(* Logix 5000 project; controller R5_CSS vendor 1 type 14 code 74 rev 19.11; software revision 19.01; part 18 of 18 *)
(* tags used below, declared in another part *)
   AlarmMasterDisable : BOOL;
   AutoTune : PIDE_AUTOTUNE;
   CSS_Heartbeat : BOOL;
   CSS_HeartbeatOffONS : BOOL;
   CSS_HeartbeatOnONS : BOOL;
   CSS_OK_TO_RUN : BOOL;   // PRU_RUN_DISABLE 0 = Cannot Run 1 = OK to Run
   CSS_Status_To_UTL_Comms : DINT;
   Fault : BOOL;
   FC101 : FLOW_CONTROL;   // QUENCH BASIN FLOW TRANSMITTER CONTROL
   FC101_Initialize : BOOL;
   FC101_Initialize_TON : TIMER;
   FC140 : FLOW_CONTROL;
   FC140A : FLOW_CONTROL;   // QUENCH TOWER UPPER SPRAY FLOW CONTROL
   FC140B : FLOW_CONTROL;   // QUENCH TOWER LOWER SPRAY FLOW CONTROL
   FC365 : FLOW_CONTROL;   // COALESCER PROCESS IMPURITY FLOW CONTROL
   FT140_TOTAL_FLOW : REAL;
   InputMax_IF8 : REAL;
   InputMin_IF8 : REAL;
   LC101 : LEVEL_CONTROL;   // QUENCH TOWER BASIN LIT
   LC101_PIDE_AUTO : BOOL;
   LC101_PIDE_CV_Hold : REAL;
   LC303A : LEVEL_CONTROL;   // AQUEOUS PHASE OF PRIMARY SETTLER
   MSG_ConnectionRateSec : DINT;
   MSG_TimeoutMultiplier : DINT;
   MSG_UnconnectedTimeoutSec : DINT;
   MyTime : DINT[10];
   P303A : PUMP_CONTROL;
   P303B : PUMP_CONTROL;
   PC132 : PRESSURE_CONTROL;
   PC132_PID : PID;
   PID_FCV365 : PID;
   PID_TCV108_Flow : PID;
   PRU_BLOWER_SEQ : INT;   // PRU BLOWER SEQUENCE NUMBER
   PRU_Quantity : DINT;
   PRU_SEQ_TMR : TIMER;   // PRU_SEQUENCE TIMER
   PRUA_READ : INT[30];
   PRUB_READ : INT[30];
   PRUC_READ : INT[30];
   PRUD_READ : INT[30];   // PRU D READ
   PRUE_READ : INT[30];
   PRUF_READ : INT[30];
   PRUG_READ : INT[30];
   PRUH_READ : INT[30];
   RandomNumber : REAL;
   RandomNumberDint : DINT;
   TC108 : TEMP_CONTROL;   // QUENCH TOWER EXIT GAS TEMPERATURE CONTROL
   TestyBit : DINT;
   TIMER : TIMER[50];   // HX A TIMER FOR START
   UTIL_1 : INT;   // ONE SHOTS FOR UTILITIES
   UTL_AlarmMaster : DINT;
   UTL_Comms : DINT[3];
   UTL_CommsLossAlm : BOOL;
   UTL_HeartbeatTimer : TIMER;
   UTL_READ_MSG : MESSAGE;
   WRS_OK : BOOL;
(* MainProgram, continued *)

ROUTINE TEMPORARY   (* ladder *)
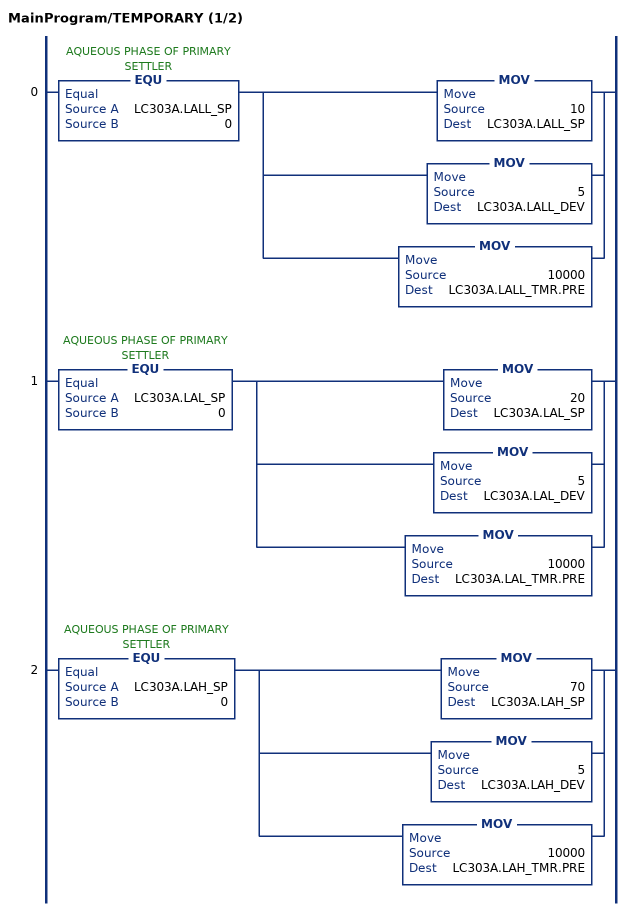
   0: EQU(LC303A.LALL_SP,0)[MOV(10,LC303A.LALL_SP) ,MOV(5,LC303A.LALL_DEV) ,MOV(10000,LC303A.LALL_TMR.PRE) ];
   1: EQU(LC303A.LAL_SP,0)[MOV(20,LC303A.LAL_SP) ,MOV(5,LC303A.LAL_DEV) ,MOV(10000,LC303A.LAL_TMR.PRE) ];
   2: EQU(LC303A.LAH_SP,0)[MOV(70,LC303A.LAH_SP) ,MOV(5,LC303A.LAH_DEV) ,MOV(10000,LC303A.LAH_TMR.PRE) ];
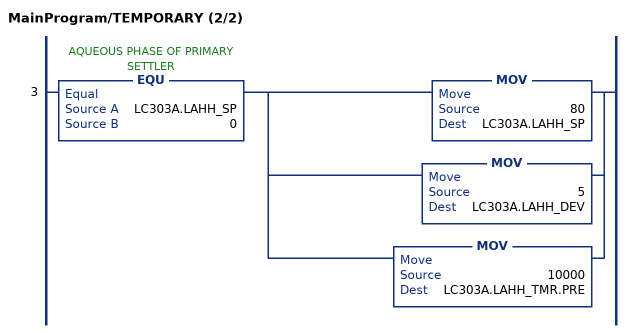
   3: EQU(LC303A.LAHH_SP,0)[MOV(80,LC303A.LAHH_SP) ,MOV(5,LC303A.LAHH_DEV) ,MOV(10000,LC303A.LAHH_TMR.PRE) ];
END_ROUTINE

ROUTINE UTIL   (* ladder *)
// UTILITIES LOGIC
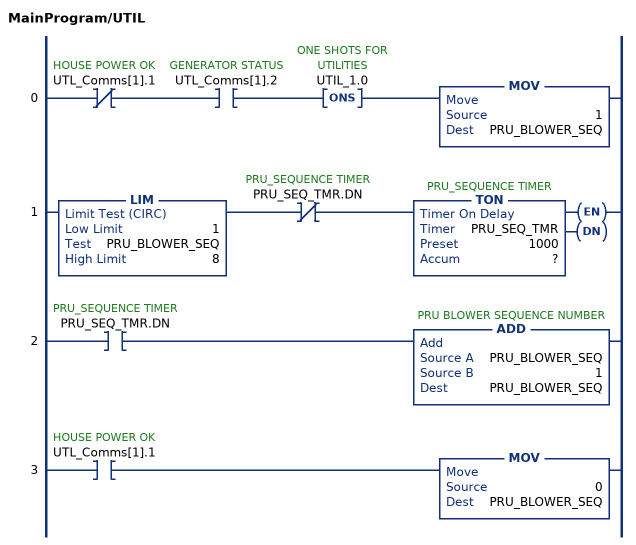
   0: XIO(UTL_Comms[1].1)XIC(UTL_Comms[1].2)ONS(UTIL_1.0)MOV(1,PRU_BLOWER_SEQ);
   1: LIM(1,PRU_BLOWER_SEQ,8)XIO(PRU_SEQ_TMR.DN)TON(PRU_SEQ_TMR,?,?);
   2: XIC(PRU_SEQ_TMR.DN)ADD(PRU_BLOWER_SEQ,1,PRU_BLOWER_SEQ);
   3: XIC(UTL_Comms[1].1)MOV(0,PRU_BLOWER_SEQ);
END_ROUTINE
END_PROGRAM

PROGRAM Never_Fault_Logic   (* main routine Main *)
VAR
   HMI_CONTROLLER_DISPLAY : MAJOR_FAULT := (TYPE := 3, CODE := 23);
   MAJORFAULT_RECORD : FAULTRECORD;
END_VAR

ROUTINE Main   (* ladder *)
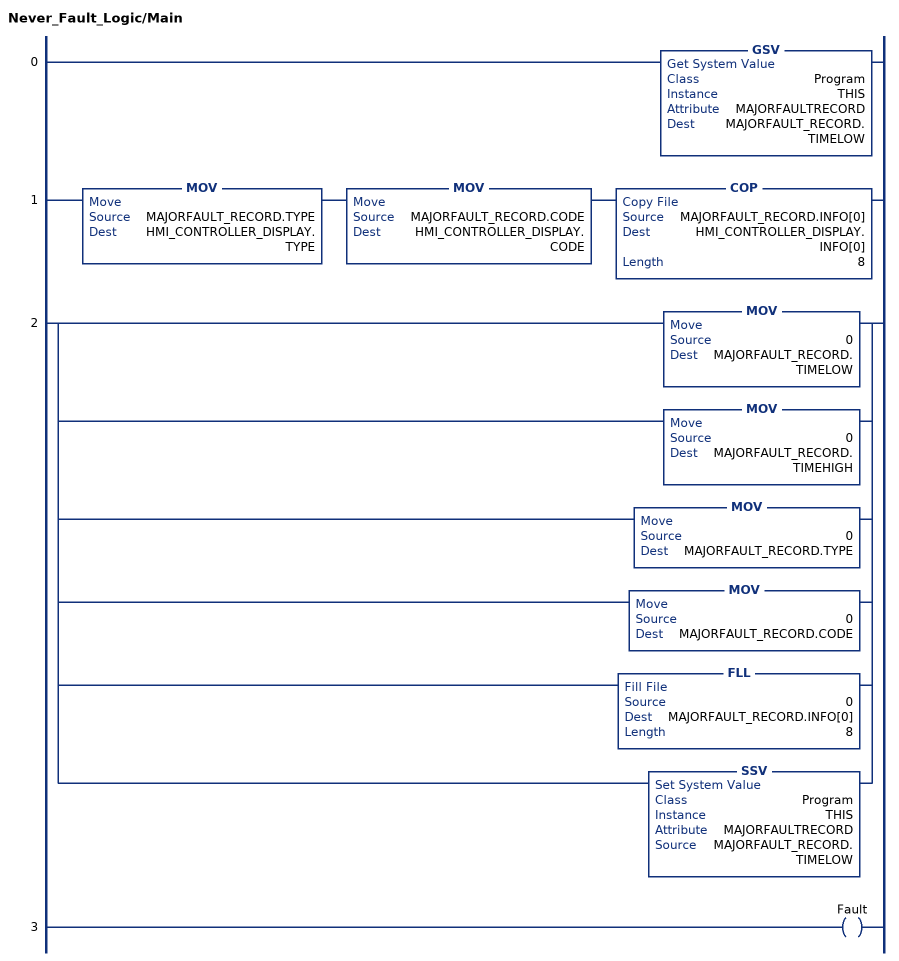
   0: GSV(Program,THIS,MAJORFAULTRECORD,MAJORFAULT_RECORD.TIMELOW);
   1: MOV(MAJORFAULT_RECORD.TYPE,HMI_CONTROLLER_DISPLAY.TYPE)MOV(MAJORFAULT_RECORD.CODE,HMI_CONTROLLER_DISPLAY.CODE)COP(MAJORFAULT_RECORD.INFO[0],HMI_CONTROLLER_DISPLAY.INFO[0],8);
   2: [MOV(0,MAJORFAULT_RECORD.TIMELOW) ,MOV(0,MAJORFAULT_RECORD.TIMEHIGH) ,MOV(0,MAJORFAULT_RECORD.TYPE) ,MOV(0,MAJORFAULT_RECORD.CODE) ,FLL(0,MAJORFAULT_RECORD.INFO[0],8) ,SSV(Program,THIS,MAJORFAULTRECORD,MAJORFAULT_RECORD.TIMELOW) ];
   3: OTE(Fault);
END_ROUTINE
END_PROGRAM

PROGRAM PIDE   (* main routine Main *)
VAR
   BNOT_01 : FBD_BOOLEAN_NOT := (Out := 1);
   BNOT_02 : FBD_BOOLEAN_NOT := (In := 1);
   SUB_01 : FBD_MATH := (SourceA := 0.049999237, SourceB := 29.966267, Dest := -29.916267);
END_VAR

ROUTINE LC101   (* function block diagram *)
   SHEET 1
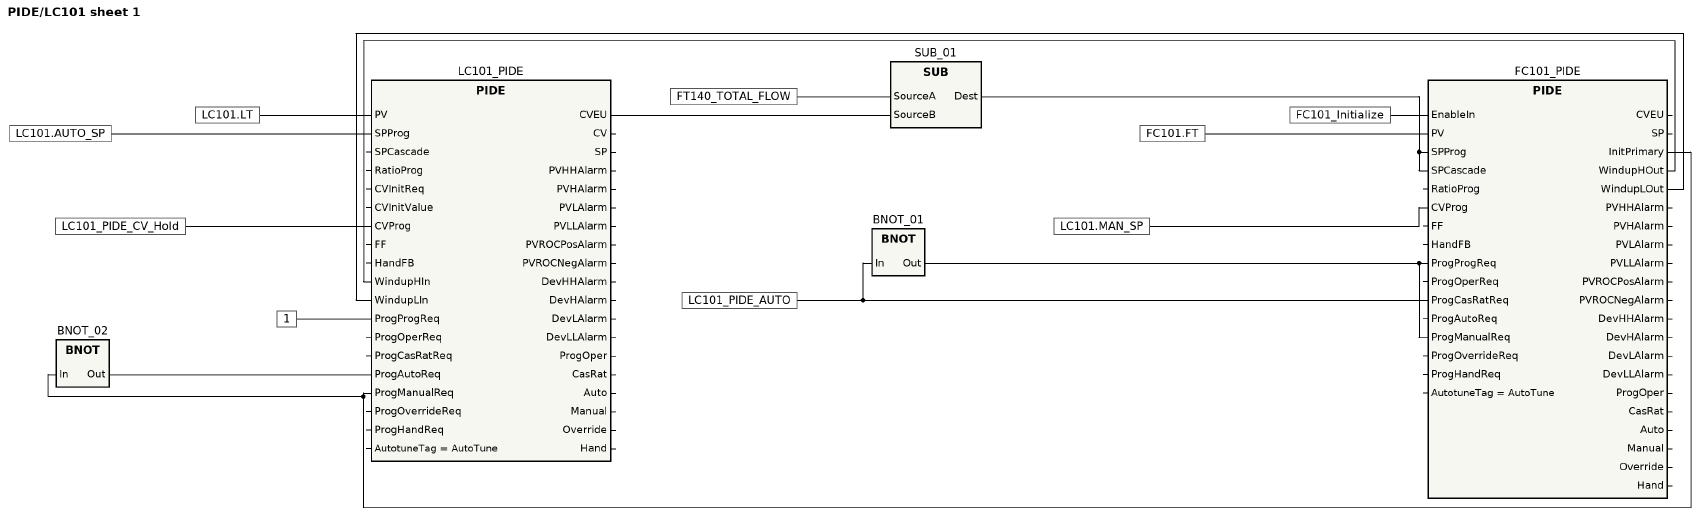
   BNOT_02 : BNOT(In := FC101_PIDE.InitPrimary {feedback});
   LC101_PIDE : PIDE(PV := LC101.LT, SPProg := LC101.AUTO_SP, CVProg := LC101_PIDE_CV_Hold, WindupHIn := FC101_PIDE.WindupHOut {feedback}, WindupLIn := FC101_PIDE.WindupLOut {feedback}, ProgProgReq := 1, ProgAutoReq := BNOT_02.Out, ProgManualReq := FC101_PIDE.InitPrimary {feedback}, AutotuneTag := AutoTune);   // unwired pins: SPCascade RatioProg CVInitReq CVInitValue FF HandFB ProgOperReq ProgCasRatReq ProgOverrideReq ProgHandReq CV SP PVHHAlarm PVHAlarm PVLAlarm PVLLAlarm PVROCPosAlarm PVROCNegAlarm DevHHAlarm DevHAlarm DevLAlarm DevLLAlarm ProgOper CasRat Auto Manual Override Hand
   BNOT_01 : BNOT(In := LC101_PIDE_AUTO);
   SUB_01 : SUB(SourceA := FT140_TOTAL_FLOW, SourceB := LC101_PIDE.CVEU);
   FC101_PIDE : PIDE(EnableIn := FC101_Initialize, PV := FC101.FT, SPProg := SUB_01.Dest, SPCascade := SUB_01.Dest, CVProg := LC101.MAN_SP, ProgProgReq := BNOT_01.Out, ProgCasRatReq := LC101_PIDE_AUTO, ProgManualReq := BNOT_01.Out, AutotuneTag := AutoTune);   // unwired pins: RatioProg FF HandFB ProgOperReq ProgAutoReq ProgOverrideReq ProgHandReq CVEU SP PVHHAlarm PVHAlarm PVLAlarm PVLLAlarm PVROCPosAlarm PVROCNegAlarm DevHHAlarm DevHAlarm DevLAlarm DevLLAlarm ProgOper CasRat Auto Manual Override Hand
END_ROUTINE

ROUTINE Main   (* ladder *)
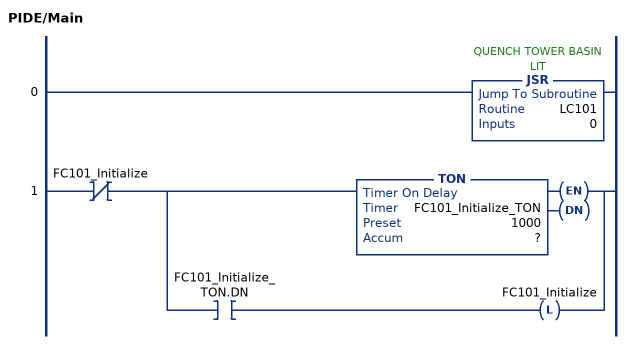
   0: JSR(LC101,0);
   1: XIO(FC101_Initialize)[TON(FC101_Initialize_TON,?,?) ,XIC(FC101_Initialize_TON.DN) OTL(FC101_Initialize) ];
END_ROUTINE
END_PROGRAM

PROGRAM POD1_MSG   (* main routine MSG *)
VAR
   PRU_BatchNewID_old : DINT[5];
END_VAR

ROUTINE MSG   (* ladder *)
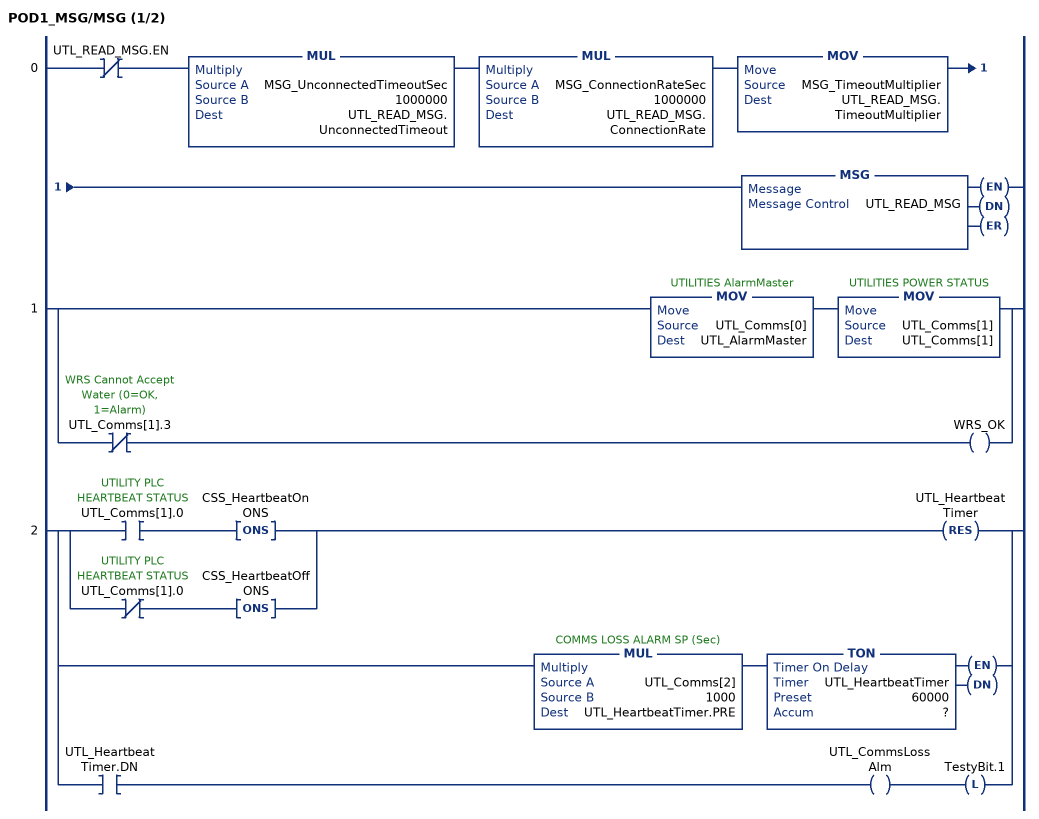
   0: XIO(UTL_READ_MSG.EN)MUL(MSG_UnconnectedTimeoutSec,1000000,UTL_READ_MSG.UnconnectedTimeout)MUL(MSG_ConnectionRateSec,1000000,UTL_READ_MSG.ConnectionRate)MOV(MSG_TimeoutMultiplier,UTL_READ_MSG.TimeoutMultiplier)MSG(UTL_READ_MSG);
   1: [MOV(UTL_Comms[0],UTL_AlarmMaster) MOV(UTL_Comms[1],UTL_Comms[1]) ,XIO(UTL_Comms[1].3) OTE(WRS_OK) ];
   2: [[XIC(UTL_Comms[1].0) ONS(CSS_HeartbeatOnONS) ,XIO(UTL_Comms[1].0) ONS(CSS_HeartbeatOffONS) ] RES(UTL_HeartbeatTimer) ,MUL(UTL_Comms[2],1000,UTL_HeartbeatTimer.PRE) TON(UTL_HeartbeatTimer,?,?) ,XIC(UTL_HeartbeatTimer.DN) OTE(UTL_CommsLossAlm) OTL(TestyBit.1) ];
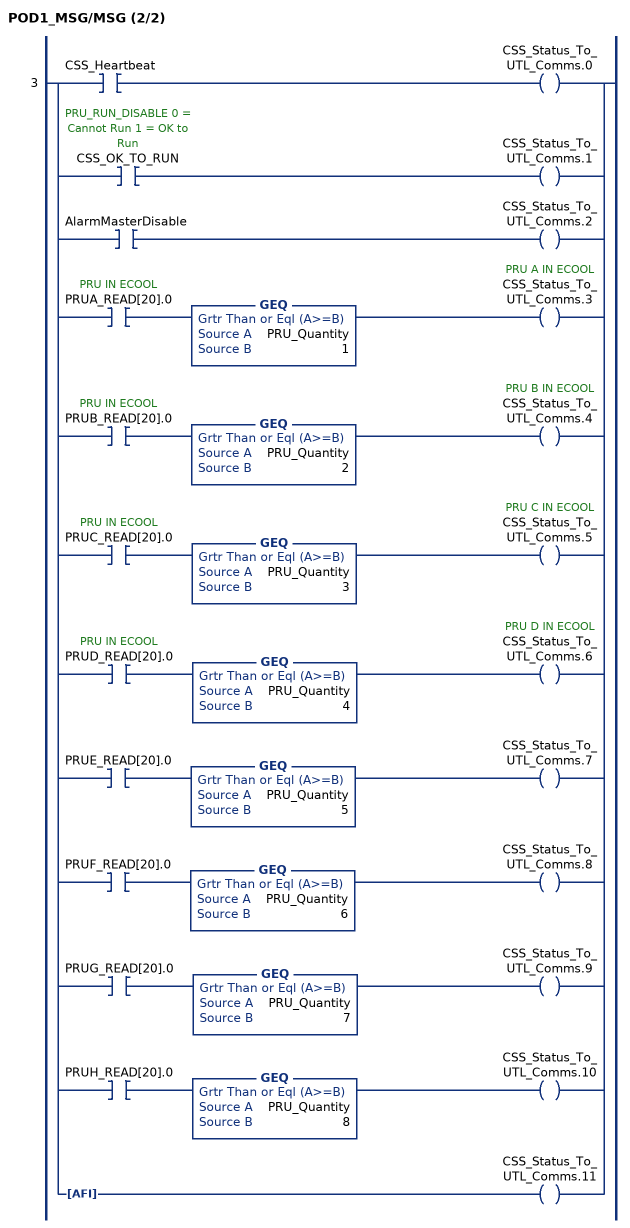
   3: [XIC(CSS_Heartbeat) OTE(CSS_Status_To_UTL_Comms.0) ,XIC(CSS_OK_TO_RUN) OTE(CSS_Status_To_UTL_Comms.1) ,XIC(AlarmMasterDisable) OTE(CSS_Status_To_UTL_Comms.2) ,XIC(PRUA_READ[20].0) GEQ(PRU_Quantity,1) OTE(CSS_Status_To_UTL_Comms.3) ,XIC(PRUB_READ[20].0) GEQ(PRU_Quantity,2) OTE(CSS_Status_To_UTL_Comms.4) ,XIC(PRUC_READ[20].0) GEQ(PRU_Quantity,3) OTE(CSS_Status_To_UTL_Comms.5) ,XIC(PRUD_READ[20].0) GEQ(PRU_Quantity,4) OTE(CSS_Status_To_UTL_Comms.6) ,XIC(PRUE_READ[20].0) GEQ(PRU_Quantity,5) OTE(CSS_Status_To_UTL_Comms.7) ,XIC(PRUF_READ[20].0) GEQ(PRU_Quantity,6) OTE(CSS_Status_To_UTL_Comms.8) ,XIC(PRUG_READ[20].0) GEQ(PRU_Quantity,7) OTE(CSS_Status_To_UTL_Comms.9) ,XIC(PRUH_READ[20].0) GEQ(PRU_Quantity,8) OTE(CSS_Status_To_UTL_Comms.10) ,AFI() OTE(CSS_Status_To_UTL_Comms.11) ];
END_ROUTINE
END_PROGRAM

PROGRAM Simulate   (* main routine MainProgram *)
VAR
   BasinFlowBalance : REAL := 94.5125;
   BasinFlowBalanceAdd : REAL := 0.45176974;
   BasinFlowBalanceAddSCLP : SCLP := (Input := 0.45176974, InputMax := 38.0, ScaledMax := 16000.0, Output := 190.21884);
   BasinFlowBalanceRawAdd : REAL := 190.21884;
   BasinFlowBalanceTmr : TIMER := (PRE := 1000);
   FC140_PID_Sim : AI_Simulate := (ControlVariable := 20.0, AI_Counts := 4038, RandomNumber := 0.939, PID_P := 1.0, PID_I := 1.0, ScaledMin := 4000, ScaledMax := 20000, PID_CV_Min := 20.0, PID_CV_Max := 100.0, UpdateSec := 1.0, DirectActing := 1);
   FC140_SUM : DINT := 4029;
   FC140_SUM_Flow : REAL := 0.36249924;
   FC140_SUM_sclp : SCLP := (Input := 4006.0, InputMin := 4000.0, InputMax := 20000.0, ScaledMax := 200.0, Output := 0.07500076);
   FC140A_Flow : REAL := 0.1449997;
   FC140A_SUM : SCLP := (Input := 0.0050003054, InputMax := 200.0, ScaledMin := 4000.0, ScaledMax := 20000.0, Output := 4000.4);
   FC140B_Flow : REAL := 0.21749955;
   FC140B_SUM : SCLP := (Input := 0.15750046, InputMax := 200.0, ScaledMin := 4000.0, ScaledMax := 20000.0, Output := 4012.6);
   FC365_FT_SIM_ENABLE : BOOL;
   FC365_PID_Sim : AI_Simulate := (ControlVariable := 50.0, AI_Counts := 12033, RandomNumber := 0.399, PID_P := 1.0, PID_I := 1.0, ScaledMin := 4000, ScaledMax := 20000, PID_CV_Max := 60.0, UpdateSec := 1.0, DirectActing := 1);
   LC101_PID_Sim : AI_Simulate := (AI_Counts := 4401, RandomNumber := 0.399, PID_P := 1.0, PID_I := 1.0, ScaledMin := 4000, ScaledMax := 20000, PID_CV_Min := 2.0, PID_CV_Max := 100.0, UpdateSec := 1.0, DirectActing := 1);
   PC132_PID_Sim : AI_Simulate := (ControlVariable := 50.0, AI_Counts := 12068, RandomNumber := 0.399, PID_P := 1.0, PID_I := 1.0, ScaledMin := 4000, ScaledMax := 20000, PID_CV_Max := 100.0, UpdateSec := 1.0);
   PC132_SIM_ENABLE : BOOL;
   TEMP_PERCENT : REAL := 50.0;
END_VAR

ROUTINE FC140   (* ladder *)
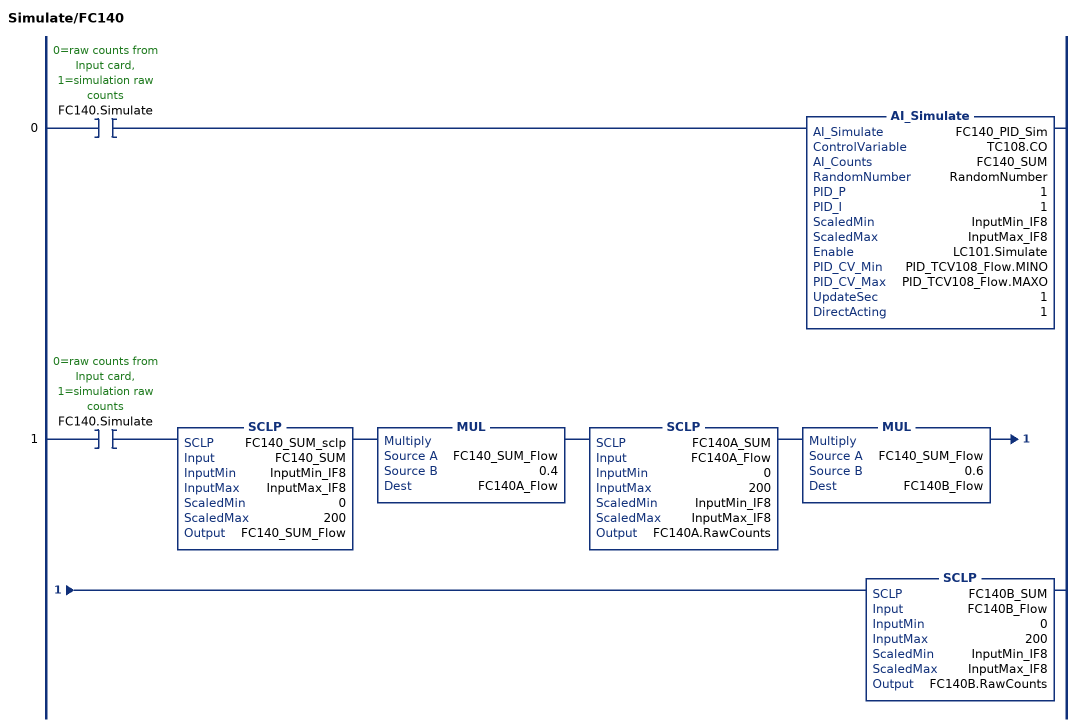
   0: XIC(FC140.Simulate)AI_Simulate(FC140_PID_Sim,TC108.CO,FC140_SUM,RandomNumber,1,1,InputMin_IF8,InputMax_IF8,LC101.Simulate,PID_TCV108_Flow.MINO,PID_TCV108_Flow.MAXO,1,1);
   1: XIC(FC140.Simulate)SCLP(FC140_SUM_sclp,FC140_SUM,InputMin_IF8,InputMax_IF8,0,200,FC140_SUM_Flow)MUL(FC140_SUM_Flow,0.4,FC140A_Flow)SCLP(FC140A_SUM,FC140A_Flow,0,200,InputMin_IF8,InputMax_IF8,FC140A.RawCounts)MUL(FC140_SUM_Flow,0.6,FC140B_Flow)SCLP(FC140B_SUM,FC140B_Flow,0,200,InputMin_IF8,InputMax_IF8,FC140B.RawCounts);
END_ROUTINE

ROUTINE FC365   (* ladder *)
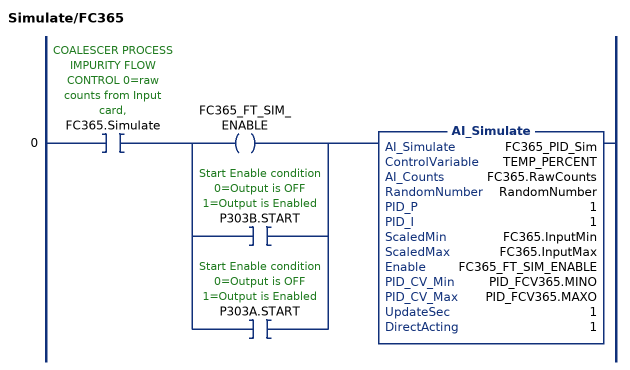
   0: XIC(FC365.Simulate)[OTE(FC365_FT_SIM_ENABLE) ,[XIC(P303B.START) ,XIC(P303A.START) ] ]AI_Simulate(FC365_PID_Sim,TEMP_PERCENT,FC365.RawCounts,RandomNumber,1,1,FC365.InputMin,FC365.InputMax,FC365_FT_SIM_ENABLE,PID_FCV365.MINO,PID_FCV365.MAXO,1,1);
END_ROUTINE

ROUTINE LC101   (* ladder *)
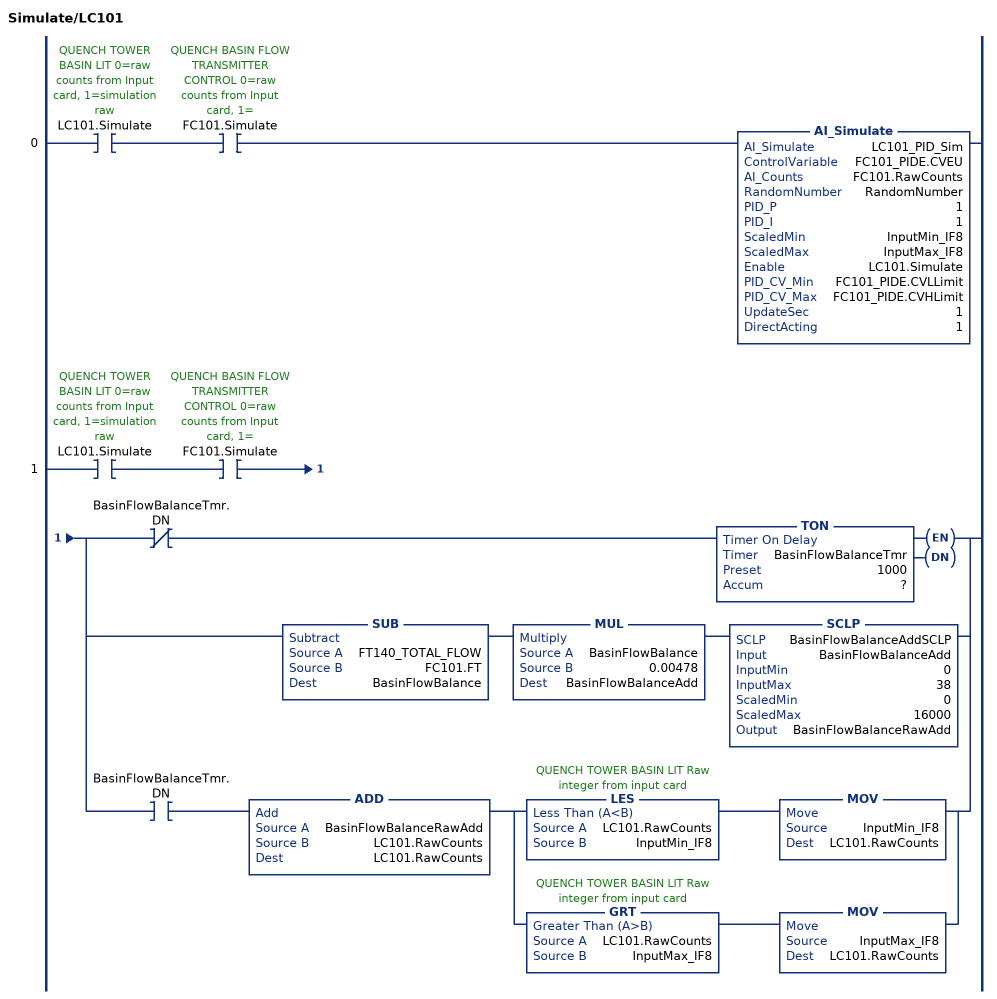
   0: XIC(LC101.Simulate)XIC(FC101.Simulate)AI_Simulate(LC101_PID_Sim,FC101_PIDE.CVEU,FC101.RawCounts,RandomNumber,1,1,InputMin_IF8,InputMax_IF8,LC101.Simulate,FC101_PIDE.CVLLimit,FC101_PIDE.CVHLimit,1,1);
   1: XIC(LC101.Simulate)XIC(FC101.Simulate)[XIO(BasinFlowBalanceTmr.DN) TON(BasinFlowBalanceTmr,?,?) ,SUB(FT140_TOTAL_FLOW,FC101.FT,BasinFlowBalance) MUL(BasinFlowBalance,0.00478,BasinFlowBalanceAdd) SCLP(BasinFlowBalanceAddSCLP,BasinFlowBalanceAdd,0,38,0,16000,BasinFlowBalanceRawAdd) ,XIC(BasinFlowBalanceTmr.DN) ADD(BasinFlowBalanceRawAdd,LC101.RawCounts,LC101.RawCounts) [LES(LC101.RawCounts,InputMin_IF8) MOV(InputMin_IF8,LC101.RawCounts) ,GRT(LC101.RawCounts,InputMax_IF8) MOV(InputMax_IF8,LC101.RawCounts) ] ];
END_ROUTINE

ROUTINE MainProgram   (* ladder *)
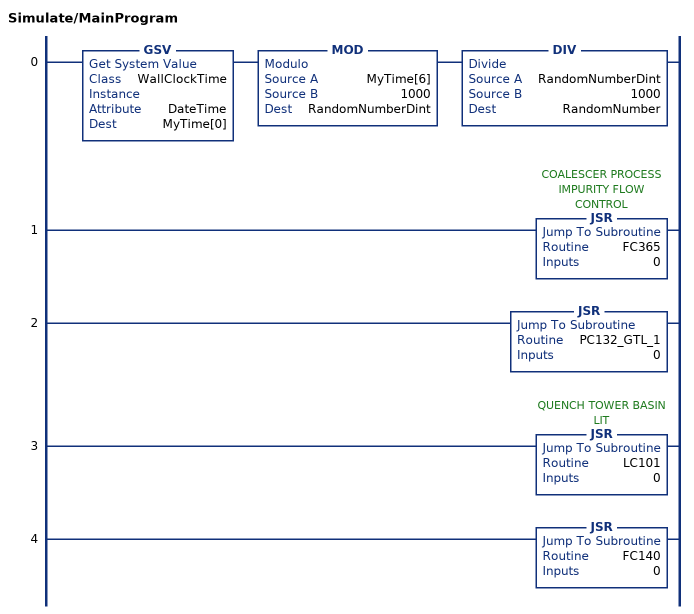
   0: GSV(WallClockTime,,DateTime,MyTime[0])MOD(MyTime[6],1000,RandomNumberDint)DIV(RandomNumberDint,1000,RandomNumber);
   1: JSR(FC365,0);
   2: JSR(PC132_GTL_1,0);
   3: JSR(LC101,0);
   4: JSR(FC140,0);
END_ROUTINE

ROUTINE PC132_GTL_1   (* ladder *)
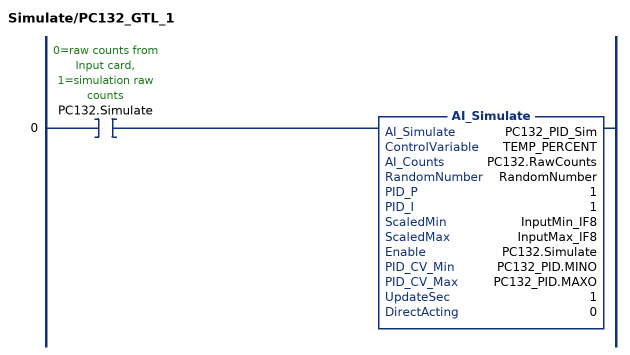
   0: XIC(PC132.Simulate)AI_Simulate(PC132_PID_Sim,TEMP_PERCENT,PC132.RawCounts,RandomNumber,1,1,InputMin_IF8,InputMax_IF8,PC132.Simulate,PC132_PID.MINO,PC132_PID.MAXO,1,0);
END_ROUTINE
END_PROGRAM
